Yaskawa INFORM job: CLAMP_GRIPPER.JBI

/JOB
//NAME CLAMP_GRIPPER
//POS
///NPOS 0,0,0,0,0,0
//INST
///DATE 2018/09/04 12:41
///ATTR SC,RW
NOP
DOUT OT#(21) OFF
DOUT OT#(20) ON
WAIT IN#(10)=ON
DOUT OT#(20) OFF
DOUT OT#(21) ON
TIMER T=0.30
DOUT OT#(21) OFF
DOUT OT#(20) ON
WAIT IN#(10)=ON
TIMER T=0.50
SET B016 1
END
